# EPICS autosave request: ADApp/Db/NDFFT_settings.req
file "NDPluginBase_settings.req", P=$(P), R=$(R)
$(P)$(R)FFTRank
$(P)$(R)FFTDirection
$(P)$(R)FFTSuppressDC
